# B&R Automation Studio project pneutrunk_plc (part 3)

#### pneutr2_reg_FF_stiff_private.h
```c
/*
 * pneutr2_reg_FF_stiff_private.h
 *
 * Academic License - for use in teaching, academic research, and meeting
 * course requirements at degree granting institutions only.  Not for
 * government, commercial, or other organizational use.
 *
 * Code generation for model "pneutr2_reg_FF_stiff".
 *
 * Model version              : 4.30
 * Simulink Coder version : 9.9 (R2023a) 19-Nov-2022
 * C source code generated on : Thu Feb 15 10:44:02 2024
 *
 * Target selection: bur_grt.tlc
 * Note: GRT includes extra infrastructure and instrumentation for prototyping
 * Embedded hardware selection: Intel->x86/Pentium
 * Code generation objectives: Unspecified
 * Validation result: Not run
 */

#ifndef RTW_HEADER_pneutr2_reg_FF_stiff_private_h_
#define RTW_HEADER_pneutr2_reg_FF_stiff_private_h_
#include "rtwtypes.h"
#include "multiword_types.h"
#include "zero_crossing_types.h"
#include "pneutr2_reg_FF_stiff.h"
#include "pneutr2_reg_FF_stiff_types.h"

extern real32_T look1_tf_binlcpw(real_T u0, const real_T bp0[], const real32_T
  table[], uint32_T maxIndex);
extern void pneutr2_reg_FF_stiff_ID1(real32_T rtu_poz_u_x, real32_T rtu_poz_u_y,
  const real_T rtu_coef_1blue[48], const real_T rtu_coef_2green[48], const
  real_T rtu_coef_3yellow[48], real32_T rtu_tuhost, B_ID1_pneutr2_reg_FF_stiff_T
  *localB);
extern void pneutr2_r_requestedalfa2deltaz1(real32_T rtu_AlphaX_ref, real32_T
  rtu_AlphaY_ref, real32_T rtu_AlphaX_real, real32_T rtu_AlphaY_real, real_T
  rtu_A, real_T rtu_B, real32_T rtu_poradie, B_requestedalfa2deltaz1_pneut_T
  *localB);
extern void pneutr2_reg_FF_s_MATLABFunction(real_T rtu_in, real_T
  rtu_previous_in, real_T rtu_step, real_T rtu_pocet_stepov, real_T rtu_last_in,
  real_T rtu_neupravujuci_uhol, B_MATLABFunction_pneutr2_reg__T *localB);

#endif                          /* RTW_HEADER_pneutr2_reg_FF_stiff_private_h_ */
```

#### pneutr2_reg_FF_stiff_types.h
```c
/*
 * pneutr2_reg_FF_stiff_types.h
 *
 * Academic License - for use in teaching, academic research, and meeting
 * course requirements at degree granting institutions only.  Not for
 * government, commercial, or other organizational use.
 *
 * Code generation for model "pneutr2_reg_FF_stiff".
 *
 * Model version              : 4.30
 * Simulink Coder version : 9.9 (R2023a) 19-Nov-2022
 * C source code generated on : Thu Feb 15 10:44:02 2024
 *
 * Target selection: bur_grt.tlc
 * Note: GRT includes extra infrastructure and instrumentation for prototyping
 * Embedded hardware selection: Intel->x86/Pentium
 * Code generation objectives: Unspecified
 * Validation result: Not run
 */

#ifndef RTW_HEADER_pneutr2_reg_FF_stiff_types_h_
#define RTW_HEADER_pneutr2_reg_FF_stiff_types_h_

/* Forward declaration for rtModel */
typedef struct tag_RTM_pneutr2_reg_FF_stiff_T RT_MODEL_pneutr2_reg_FF_stiff_T;

#endif                            /* RTW_HEADER_pneutr2_reg_FF_stiff_types_h_ */
```

#### rt_nonfinite.h
```c
/*
 * rt_nonfinite.h
 *
 * Academic License - for use in teaching, academic research, and meeting
 * course requirements at degree granting institutions only.  Not for
 * government, commercial, or other organizational use.
 *
 * Code generation for model "pneutr2_reg_FF_stiff".
 *
 * Model version              : 4.30
 * Simulink Coder version : 9.9 (R2023a) 19-Nov-2022
 * C source code generated on : Thu Feb 15 10:44:02 2024
 *
 * Target selection: bur_grt.tlc
 * Note: GRT includes extra infrastructure and instrumentation for prototyping
 * Embedded hardware selection: Intel->x86/Pentium
 * Code generation objectives: Unspecified
 * Validation result: Not run
 */

#ifndef RTW_HEADER_rt_nonfinite_h_
#define RTW_HEADER_rt_nonfinite_h_
#include <stddef.h>
#include "rtwtypes.h"
#define NOT_USING_NONFINITE_LITERALS   1

extern real_T rtInf;
extern real_T rtMinusInf;
extern real_T rtNaN;
extern real32_T rtInfF;
extern real32_T rtMinusInfF;
extern real32_T rtNaNF;
extern void rt_InitInfAndNaN(size_t realSize);
extern boolean_T rtIsInf(real_T value);
extern boolean_T rtIsInfF(real32_T value);
extern boolean_T rtIsNaN(real_T value);
extern boolean_T rtIsNaNF(real32_T value);
typedef struct {
  struct {
    uint32_T wordH;
    uint32_T wordL;
  } words;
} BigEndianIEEEDouble;

typedef struct {
  struct {
    uint32_T wordL;
    uint32_T wordH;
  } words;
} LittleEndianIEEEDouble;

typedef struct {
  union {
    real32_T wordLreal;
    uint32_T wordLuint;
  } wordL;
} IEEESingle;

#endif                                 /* RTW_HEADER_rt_nonfinite_h_ */
```

#### rtGetNaN.h
```c
/*
 * rtGetNaN.h
 *
 * Academic License - for use in teaching, academic research, and meeting
 * course requirements at degree granting institutions only.  Not for
 * government, commercial, or other organizational use.
 *
 * Code generation for model "pneutr2_reg_FF_stiff".
 *
 * Model version              : 4.30
 * Simulink Coder version : 9.9 (R2023a) 19-Nov-2022
 * C source code generated on : Thu Feb 15 10:44:02 2024
 *
 * Target selection: bur_grt.tlc
 * Note: GRT includes extra infrastructure and instrumentation for prototyping
 * Embedded hardware selection: Intel->x86/Pentium
 * Code generation objectives: Unspecified
 * Validation result: Not run
 */

#ifndef RTW_HEADER_rtGetNaN_h_
#define RTW_HEADER_rtGetNaN_h_
#include "rt_nonfinite.h"
#include "rtwtypes.h"

extern real_T rtGetNaN(void);
extern real32_T rtGetNaNF(void);

#endif                                 /* RTW_HEADER_rtGetNaN_h_ */
```

#### rtGetNaN.c
```c
/*
 * rtGetNaN.c
 *
 * Academic License - for use in teaching, academic research, and meeting
 * course requirements at degree granting institutions only.  Not for
 * government, commercial, or other organizational use.
 *
 * Code generation for model "pneutr2_reg_FF_stiff".
 *
 * Model version              : 4.30
 * Simulink Coder version : 9.9 (R2023a) 19-Nov-2022
 * C source code generated on : Thu Feb 15 10:44:02 2024
 *
 * Target selection: bur_grt.tlc
 * Note: GRT includes extra infrastructure and instrumentation for prototyping
 * Embedded hardware selection: Intel->x86/Pentium
 * Code generation objectives: Unspecified
 * Validation result: Not run
 */

#include "rtwtypes.h"
#include "rtGetNaN.h"
#include <stddef.h>
#include "rt_nonfinite.h"
#define NumBitsPerChar                 8U

/*
 * Initialize rtNaN needed by the generated code.
 * NaN is initialized as non-signaling. Assumes IEEE.
 */
real_T rtGetNaN(void)
{
  size_t bitsPerReal = sizeof(real_T) * (NumBitsPerChar);
  real_T nan = 0.0;
  if (bitsPerReal == 32U) {
    nan = rtGetNaNF();
  } else {
    uint16_T one = 1U;
    enum {
      LittleEndian,
      BigEndian
    } machByteOrder = (*((uint8_T *) &one) == 1U) ? LittleEndian : BigEndian;
    switch (machByteOrder) {
     case LittleEndian:
      {
        union {
          LittleEndianIEEEDouble bitVal;
          real_T fltVal;
        } tmpVal;

        tmpVal.bitVal.words.wordH = 0xFFF80000U;
        tmpVal.bitVal.words.wordL = 0x00000000U;
        nan = tmpVal.fltVal;
        break;
      }

     case BigEndian:
      {
        union {
          BigEndianIEEEDouble bitVal;
          real_T fltVal;
        } tmpVal;

        tmpVal.bitVal.words.wordH = 0x7FFFFFFFU;
        tmpVal.bitVal.words.wordL = 0xFFFFFFFFU;
        nan = tmpVal.fltVal;
        break;
      }
    }
  }

  return nan;
}

/*
 * Initialize rtNaNF needed by the generated code.
 * NaN is initialized as non-signaling. Assumes IEEE.
 */
real32_T rtGetNaNF(void)
{
  IEEESingle nanF = { { 0.0F } };

  uint16_T one = 1U;
  enum {
    LittleEndian,
    BigEndian
  } machByteOrder = (*((uint8_T *) &one) == 1U) ? LittleEndian : BigEndian;
  switch (machByteOrder) {
   case LittleEndian:
    {
      nanF.wordL.wordLuint = 0xFFC00000U;
      break;
    }

   case BigEndian:
    {
      nanF.wordL.wordLuint = 0x7FFFFFFFU;
      break;
    }
  }

  return nanF.wordL.wordLreal;
}
```

### Types.typ
```iecst
TYPE
	mech : 	STRUCT
		pozadovany_uhol_y_old : ARRAY[0..6]OF REAL;
		real_uhol_y_kalibrovane : ARRAY[0..6]OF REAL;
		real_uhol_x_kalibrovane : ARRAY[0..6]OF REAL;
		pozadovany_uhol_y : ARRAY[0..6]OF REAL;
		pozadovany_uhol_x : ARRAY[0..6]OF REAL;
		FF_stiffness : ARRAY[0..6]OF REAL;
		PID_P : ARRAY[0..6]OF REAL;
		PID_I : ARRAY[0..6]OF REAL;
		PID_D : ARRAY[0..6]OF REAL;
		PID_N : ARRAY[0..6]OF REAL;
		reset_I_reg : ARRAY[0..6]OF REAL;
		tlak3 : ARRAY[0..6]OF REAL;
		tlak2 : ARRAY[0..6]OF REAL;
		tlak1 : ARRAY[0..6]OF REAL;
		poradie : ARRAY[0..6]OF INT;
		error_total : ARRAY[0..6]OF REAL;
		error_y : ARRAY[0..6]OF REAL;
		error_x : ARRAY[0..6]OF REAL;
		pozadovany_uhol_x_old : ARRAY[0..6]OF REAL;
		nula_y : ARRAY[0..6]OF REAL;
		nula_x : ARRAY[0..6]OF REAL;
		pozadovanyLinear : REAL;
		efektor : BOOL;
	END_STRUCT;
END_TYPE
```

### mem_mgr.h
```c
/*
 * Copyright 1994-2002 The MathWorks, Inc.
 *
 * File: mem_mgr.h
 *
 * Abstract:
 */

#ifndef __MEM_MGR__
#define __MEM_MGR__

struct MemBufHdr {
    struct MemBufHdr *memBufNext;
    struct MemBufHdr *memBufPrev;
    char   *MemBuf;
    int    size;
};

typedef struct MemBufHdr MemBufHdr;

extern void ExtModeFree(void *mem);

extern void *ExtModeMalloc(size_t size);

extern void *ExtModeCalloc(size_t number, size_t size);

#endif /* __MEM_MGR__ */

/* [EOF] mem_mgr.h */
```

### Program Logical/Source/Narazy

#### Cyclic.st
```iecst
PROGRAM _CYCLIC

	FOR i:=0 TO 6 BY 1 DO
		IF modul.naraz[i] = TRUE THEN
			modul.narazAktivny	:= TRUE;
			step				:= 5;
		END_IF
	END_FOR

END_PROGRAM
```

### Program Logical/Source/RS485/Receiver

#### Receiver.typ
```iecst
(********************************************************************
 * COPYRIGHT -- Bernecker + Rainer
 ********************************************************************
 * Program: Receiver
 * File: Receiver.typ
 * Author: Bernecker & Rainer
 * Created: January 25, 2010
 ********************************************************************
 * Local data types of program Receiver
 ********************************************************************)
(*Enumeration for Statemachine*)

TYPE
	enRECV_STEPS :
		(
		FRM_WAIT := 0, (*Defines the wait step*)
		FRM_OPEN, (*Defines Step for FRM_xopen() *)
		FRM_READ, (*Defines Step for FRM_read()*)
		FRM_COPY_RD_DATA, (*Defines Step for storing read data*)
		FRM_RBUF, (*Defines Step for FRM_rbuf()*)
		FRM_CLOSE, (*Defines Step for FRM_close()*)
		FRM_ERROR := 255 (*Defines Step for Errorhandling*)
		);
END_TYPE

(*Command data type*)

TYPE
	command_typ : 	STRUCT
		open_receive : BOOL; (*Open serial port and receive data*)
		close : BOOL; (*Close serial port*)
	END_STRUCT;
END_TYPE

(*Receiver type*)

TYPE
	Receiver_typ : 	STRUCT
		step : enRECV_STEPS; (*Step of the Statemachine*)
		Commands : command_typ; (*Commandinterface*)
		receive_data : ARRAY[0..10]OF BYTE; (*receive data*)
		FRM_xopen_0 : FRM_xopen; (*Functionblock FRM_xopen()*)
		xopenConfig : XOPENCONFIG; (*Configuration Type for FRM_xopen()*)
		FRM_read_0 : FRM_read; (*Functionblock FRM_read()*)
		FRM_rbuf_0 : FRM_rbuf; (*Functionblock FRM_rbuf()*)
		FRM_close_0 : FRM_close; (*Functionblock FRM_close()*)
	END_STRUCT;
END_TYPE
```

#### ReceiverCyclic.st
```iecst
(********************************************************************
 * COPYRIGHT -- Bernecker + Rainer
 ********************************************************************
 * Program: Receiver
 * File: ReceiverCyclic.st
 * Author: Bernecker & Rainer
 * Created: January 25, 2010
 ********************************************************************
 * Implementation of program Receiver
 ********************************************************************)

(*************init program**********************)
PROGRAM _INIT
	Receiver.Commands.open_receive := TRUE;												(*enable Receiver by default*)
END_PROGRAM

(*************cyclic program********************)
PROGRAM _CYCLIC

	CASE Receiver.step OF
		FRM_WAIT:	(*--- wait for command*)

			IF Receiver.Commands.open_receive = TRUE THEN								(*command for Receiver activation*)
				Receiver.step := FRM_OPEN;
   			END_IF

			(*close will be requested in step FRM_RBUF*)

		FRM_OPEN:	(*--- open serial interface*)

			(*Parameters for FRM_xopen()*)
			Receiver.FRM_xopen_0.enable := TRUE;
			Receiver.FRM_xopen_0.device := ADR('IF6.ST1.IF1');							(*Devicename --> see your serial interface properties*)
			Receiver.FRM_xopen_0.mode := ADR('/PHY=RS485 /BD=38400 /DB=8 /PA=N /SB=1'); (*Modestring --> specifies the seria operation mode*)
			Receiver.FRM_xopen_0.config := ADR(Receiver.xopenConfig) ;					(*Additional Parameters, optional*)

			(*Additional Parameters for FRM_xopen()*)
			Receiver.xopenConfig.idle := 10;											(*Idle time between two characters*)
			Receiver.xopenConfig.delimc := 0;											(*activate two delimeters*)
			Receiver.xopenConfig.delim[0] := 0; 										(*e.g. CR - carridge return -> dec 13*)
			Receiver.xopenConfig.delim[1] := 0; 										(*e.g. LF - line feed -> dec 10*)
			Receiver.xopenConfig.tx_cnt := 3;											(*number of transmit buffers*)
			Receiver.xopenConfig.rx_cnt := 3; 											(*number of receive buffers*)
			Receiver.xopenConfig.tx_len := 256; 										(*length of transmit buffers*)
			Receiver.xopenConfig.rx_len := 256; 										(*lenght of receive buffers*)
			Receiver.xopenConfig.argc := 0;												(*activate additional options*)
			Receiver.xopenConfig.argv := 0;												(*parameters for additional options (check help)*)

			Receiver.FRM_xopen_0();														(*call the FRM_xopen() function*)

			IF Receiver.FRM_xopen_0.status = 0 THEN
				Receiver.step := FRM_READ;												(*Interface opend successfully --> next step*)
			ELSIF Receiver.FRM_xopen_0.status = BUSY THEN
				Receiver.step := FRM_OPEN;												(*operation not finished yet --> call again*)
			ELSE
				Receiver.step := FRM_ERROR;												(*function returned errorcode --> check help*)
   			END_IF

		FRM_READ:	(*--- read data from serial interface*)
			Receiver.FRM_read_0.enable := TRUE;
   			Receiver.FRM_read_0.ident := Receiver.FRM_xopen_0.ident;

			Receiver.FRM_read_0();														(*call the FRM_read() function*)

			IF Receiver.FRM_read_0.status = 0 THEN
				Receiver.step := FRM_COPY_RD_DATA;										(*system returned a valid data --> next step*)
			ELSIF Receiver.FRM_read_0.status = frmERR_NOINPUT THEN
				Receiver.step := FRM_READ;												(*no data available --> call again*)
			ELSIF Receiver.FRM_read_0.status = frmERR_INPUTERROR THEN
				Receiver.step := FRM_RBUF;												(*received Frame with defective characters, skip data*)
			ELSE
				Receiver.step := FRM_ERROR;												(*function returned errorcode --> check help*)
   			END_IF

		FRM_COPY_RD_DATA: (*--- copy data out of the receive buffer*)
			(*
			FOR i:=0 TO 8 BY 1 DO
				packet485.packet[i] := Receiver.receive_data[i];
			END_FOR
			*)
			memset(ADR(Receiver.receive_data),0,SIZEOF(Receiver.receive_data));			(*clear read_data buffer*)
			memcpy(ADR(Receiver.receive_data),Receiver.FRM_read_0.buffer,Receiver.FRM_read_0.buflng);     (*copy and evaluate read data*)

			IF(Receiver.receive_data[0] = 255)THEN
				IF(Receiver.receive_data[1] = 255)THEN
					IF(Receiver.receive_data[9] = 254)THEN
						IF(Receiver.receive_data[10] = 254)THEN
							IF(Receiver.receive_data[2] = 1)THEN
								modul.uholINT1 := BYTE_TO_INT(Receiver.receive_data[5]);
								modul.uholINT1 := SHL(modul.uholINT1,8);
								modul.uholINT1  := modul.uholINT1  + BYTE_TO_INT(Receiver.receive_data[6]);
								modul.uhol1[0] := modul.uholINT1;
								modul.uhol1[0] := modul.uhol1[0]*260/1024 - 130;
								modul.uhol1[0] := modul.uhol1[0]*1.0254 + 88.307;
								modul.uholINT2 := BYTE_TO_INT(Receiver.receive_data[7]);
								modul.uholINT2 := SHL(modul.uholINT2,8);
								modul.uholINT2  := modul.uholINT2  + BYTE_TO_INT(Receiver.receive_data[8]);
								modul.uhol2[0] := (modul.uholINT2);
								modul.uhol2[0] := modul.uhol2[0]*260/1024 - 130;
								modul.uhol2[0] := modul.uhol2[0]*1.0254 + 88.307;
							ELSIF(Receiver.receive_data[2] = 2)THEN
								modul.uholINT1 := BYTE_TO_INT(Receiver.receive_data[5]);
								modul.uholINT1 := SHL(modul.uholINT1,8);
								modul.uholINT1  := modul.uholINT1  + BYTE_TO_INT(Receiver.receive_data[6]);
								modul.uhol1[1] := (modul.uholINT1);
								modul.uhol1[1] := modul.uhol1[1]*260/1024 - 130;
								modul.uhol1[1] := modul.uhol1[1]*1.0254 + 88.307;
								modul.uholINT2 := BYTE_TO_INT(Receiver.receive_data[7]);
								modul.uholINT2 := SHL(modul.uholINT2,8);
								modul.uholINT2  := modul.uholINT2  + BYTE_TO_INT(Receiver.receive_data[8]);
								modul.uhol2[1] := (modul.uholINT2);
								modul.uhol2[1] := modul.uhol2[1]*260/1024 - 130;
								modul.uhol2[1] := modul.uhol2[1]*1.0254 + 88.307;
							ELSIF(Receiver.receive_data[2] = 3)THEN
								modul.uholINT1 := BYTE_TO_INT(Receiver.receive_data[5]);
								modul.uholINT1 := SHL(modul.uholINT1,8);
								modul.uholINT1  := modul.uholINT1  + BYTE_TO_INT(Receiver.receive_data[6]);
								modul.uhol1[2] := (modul.uholINT1);
								modul.uhol1[2] := modul.uhol1[2]*260/1024 - 130;
								modul.uhol1[2] := modul.uhol1[2]*1.0254 + 88.307;
								modul.uholINT2 := BYTE_TO_INT(Receiver.receive_data[7]);
								modul.uholINT2 := SHL(modul.uholINT2,8);
								modul.uholINT2  := modul.uholINT2  + BYTE_TO_INT(Receiver.receive_data[8]);
								modul.uhol2[2] := (modul.uholINT2);
								modul.uhol2[2] := modul.uhol2[2]*260/1024 - 130;
								modul.uhol2[2] := modul.uhol2[2]*1.0254 + 88.307;
								IF Receiver.receive_data[4] = 3 THEN
									modul.naraz[2]	:= TRUE;
								ELSE
									modul.naraz[2]	:= FALSE;
								END_IF
							ELSIF(Receiver.receive_data[2] = 4)THEN
								modul.uholINT1 := BYTE_TO_INT(Receiver.receive_data[5]);
								modul.uholINT1 := SHL(modul.uholINT1,8);
								modul.uholINT1  := modul.uholINT1  + BYTE_TO_INT(Receiver.receive_data[6]);
								modul.uhol1[3] := (modul.uholINT1);
								modul.uhol1[3] := modul.uhol1[3]*260/1024 - 130;
								modul.uhol1[3] := modul.uhol1[3]*1.0254 + 88.307;
								modul.uholINT2 := BYTE_TO_INT(Receiver.receive_data[7]);
								modul.uholINT2 := SHL(modul.uholINT2,8);
								modul.uholINT2  := modul.uholINT2  + BYTE_TO_INT(Receiver.receive_data[8]);
								modul.uhol2[3] := (modul.uholINT2);
								modul.uhol2[3] := modul.uhol2[3]*260/1024 - 130;
								modul.uhol2[3] := modul.uhol2[3]*1.0254 + 88.307;
								IF Receiver.receive_data[4] = 3 THEN
									modul.naraz[3]	:= TRUE;
								ELSE
									modul.naraz[3]	:= FALSE;
								END_IF
							ELSIF(Receiver.receive_data[2] = 5)THEN
								modul.uholINT1 := BYTE_TO_INT(Receiver.receive_data[5]);
								modul.uholINT1 := SHL(modul.uholINT1,8);
								modul.uholINT1  := modul.uholINT1  + BYTE_TO_INT(Receiver.receive_data[6]);
								modul.uhol1[4] := (modul.uholINT1);
								modul.uhol1[4] := modul.uhol1[4]*260/1024 - 130;
								modul.uhol1[4] := modul.uhol1[4]*1.0254 + 88.307;
								modul.uholINT2 := BYTE_TO_INT(Receiver.receive_data[7]);
								modul.uholINT2 := SHL(modul.uholINT2,8);
								modul.uholINT2  := modul.uholINT2  + BYTE_TO_INT(Receiver.receive_data[8]);
								modul.uhol2[4] := (modul.uholINT2);
								modul.uhol2[4] := modul.uhol2[4]*260/1024 - 130;
								modul.uhol2[4] := modul.uhol2[4]*1.0254 + 88.307;
								IF Receiver.receive_data[4] = 3 THEN
									modul.naraz[4]	:= TRUE;
								ELSE
									modul.naraz[4]	:= FALSE;
								END_IF
							ELSIF(Receiver.receive_data[2] = 6)THEN
								modul.uholINT1 := BYTE_TO_INT(Receiver.receive_data[5]);
								modul.uholINT1 := SHL(modul.uholINT1,8);
								modul.uholINT1  := modul.uholINT1  + BYTE_TO_INT(Receiver.receive_data[6]);
								modul.uhol1[5] := (modul.uholINT1);
								modul.uhol1[5] := modul.uhol1[5]*260/1024 - 130;
								modul.uhol1[5] := modul.uhol1[5]*1.0254 + 88.307;
								modul.uholINT2 := BYTE_TO_INT(Receiver.receive_data[7]);
								modul.uholINT2 := SHL(modul.uholINT2,8);
								modul.uholINT2  := modul.uholINT2  + BYTE_TO_INT(Receiver.receive_data[8]);
								modul.uhol2[5] := (modul.uholINT2);
								modul.uhol2[5] := modul.uhol2[5]*260/1024 - 130;
								modul.uhol2[5] := modul.uhol2[5]*1.0254 + 88.307;
								IF Receiver.receive_data[4] = 3 THEN
									modul.naraz[5]	:= TRUE;
								ELSE
									modul.naraz[5]	:= FALSE;
								END_IF
							ELSIF(Receiver.receive_data[2] = 7)THEN
								modul.uholINT1 := BYTE_TO_INT(Receiver.receive_data[5]);
								modul.uholINT1 := SHL(modul.uholINT1,8);
								modul.uholINT1  := modul.uholINT1  + BYTE_TO_INT(Receiver.receive_data[6]);
								modul.uhol1[6] := (modul.uholINT1);
								modul.uhol1[6] := modul.uhol1[6]*260/1024 - 130;
								modul.uhol1[6] := modul.uhol1[6]*1.0254 + 88.307;
								modul.uholINT2 := BYTE_TO_INT(Receiver.receive_data[7]);
								modul.uholINT2 := SHL(modul.uholINT2,8);
								modul.uholINT2  := modul.uholINT2  + BYTE_TO_INT(Receiver.receive_data[8]);
								modul.uhol2[6] := (modul.uholINT2);
								modul.uhol2[6] := modul.uhol2[6]*260/1024 - 130;
								modul.uhol2[6] := modul.uhol2[6]*1.0254 + 88.307;
								IF Receiver.receive_data[4] = 1 OR Receiver.receive_data[4] = 2 THEN //lebo dve moduly su zapojene do jednej dosky
									modul.naraz[6]	:= TRUE;
								ELSE
									modul.naraz[6]	:= FALSE;
								END_IF
							ELSIF(Receiver.receive_data[2] = 8)THEN
								IF Receiver.receive_data[4] = 3 THEN
									modul.naraz[7]	:= TRUE;
								ELSE
									modul.naraz[7]	:= FALSE;
								END_IF
							END_IF
						END_IF
					END_IF
				END_IF
			END_IF

			Receiver.step := FRM_RBUF;													(*release read buffer*)

		FRM_RBUF:	(*--- release readbuffer*)

			(*Parameters for FRM_rbuf()*)
			Receiver.FRM_rbuf_0.enable := TRUE;
			Receiver.FRM_rbuf_0.ident := Receiver.FRM_xopen_0.ident;					(*ident from FRM_xopen()*)
			Receiver.FRM_rbuf_0.buffer := Receiver.FRM_read_0.buffer;					(*read buffer*)
			Receiver.FRM_rbuf_0.buflng := Receiver.FRM_read_0.buflng;					(*length of sendbuffer*)

			Receiver.FRM_rbuf_0();														(*call the FRM_rbuf() function*)

			IF Receiver.FRM_rbuf_0.status = 0 THEN
				IF Receiver.Commands.close = TRUE THEN
					Receiver.Commands.open_receive := FALSE;								(*disable command open_send*)
					Receiver.step := FRM_CLOSE;											(*request to close serial port*)
				ELSE
					Receiver.step := FRM_READ;											(*read again*)
				END_IF
			ELSIF Receiver.FRM_rbuf_0.status = BUSY THEN
				Receiver.step := FRM_RBUF;												(*operation not finished yet --> call again*)
			ELSIF Receiver.FRM_rbuf_0.status = frmERR_INVALIDBUFFER THEN
				Receiver.step := FRM_READ;												(*buffer is invalid --> read again*)
			ELSE
				Receiver.step := FRM_ERROR;												(*function returned errorcode --> check help*)
   			END_IF

		FRM_CLOSE:	(*--- close the interface*)
			Receiver.FRM_close_0.enable := TRUE;
   			Receiver.FRM_close_0.ident := Receiver.FRM_xopen_0.ident;					(*ident from FRM_xopen()*)

			Receiver.FRM_close_0();														(*call the FRM_close() function*)

			IF Receiver.FRM_close_0.status = 0 THEN
				Receiver.Commands.close := FALSE;										(*disable close command*)
				Receiver.step := FRM_WAIT;												(*closed interface successfully --> wait step*)
			ELSIF Receiver.FRM_close_0.status = BUSY THEN
				Receiver.step := FRM_CLOSE;												(*operation not finished yet --> call again*)
			ELSE
				Receiver.step := FRM_ERROR;												(*function returned errorcode --> check help*)
			END_IF

		FRM_ERROR:	(*--- error handling*)
			; (*not implementet yet, check help for error codes*)
 	END_CASE

END_PROGRAM
```

### Program Logical/Source/RS485/Sender

#### SenderCyclic.st
```iecst
(********************************************************************
 * COPYRIGHT -- Bernecker + Rainer
 ********************************************************************
 * Program: Sender
 * File: SenderCyclic.st
 * Author: Bernecker & Rainer
 * Created: January 25, 2010
 ********************************************************************
 * Implementation of program Sender
 ********************************************************************)

(*************init program**********************)
PROGRAM _INIT
	Sender.Commands.open_send := TRUE;												(*enable sender by default*)
	packet485.sendPacketFinal[0] := 255;
	packet485.sendPacketFinal[1] := 255;
	packet485.sendPacketFinal[2] := 1;				// ID
	packet485.sendPacketFinal[3] := 1;
	packet485.sendPacketFinal[4] := 254;
	packet485.sendPacketFinal[5] := 254;
	Sender.step					 := FRM_WAIT;
END_PROGRAM

(*************cyclic program********************)
PROGRAM _CYCLIC

	CASE Sender.step OF
		FRM_WAIT:	(*--- wait for command*)

			IF Sender.Commands.open_send = TRUE THEN								(*command for sender activation*)
				Sender.step := FRM_OPEN;
   			END_IF

			(*close will be requested in step FRM_WRITE*)

		FRM_OPEN:	(*--- open serial interface*)

			(*Parameters for FRM_xopen()*)
			Sender.FRM_xopen_0.enable := TRUE;
			Sender.FRM_xopen_0.device := ADR('IF6.ST1.IF1');										(*Devicename --> see your serial interface properties*)
			Sender.FRM_xopen_0.mode := ADR('/PHY=RS485 /BD=38400 /DB=8 /PA=N /SB=1'); 		(*Modestring --> specifies the seria operation mode*)
			Sender.FRM_xopen_0.config := ADR(Sender.xopenConfig) ;					(*Additional Parameters, optional*)

			(*Additional Parameters for FRM_xopen()*)
			Sender.xopenConfig.idle := 10;											(*Idle time between two characters*)
			Sender.xopenConfig.delimc := 0;											(*activate two delimeters*)
			Sender.xopenConfig.delim[0] := 0; 										(*CR - carridge return -> dec 13*)
			Sender.xopenConfig.delim[1] := 0; 										(*LF - line feed -> dec 10*)
			Sender.xopenConfig.tx_cnt := 3;											(*number of transmit buffers*)
			Sender.xopenConfig.rx_cnt := 3; 										(*number of receive buffers*)
			Sender.xopenConfig.tx_len := 256; 										(*length of transmit buffers*)
			Sender.xopenConfig.rx_len := 256; 										(*lenght of receive buffers*)
			Sender.xopenConfig.argc := 0;											(*activate additional options*)
			Sender.xopenConfig.argv := 0;											(*parameters for additional options (check help)*)

			Sender.FRM_xopen_0();													(*call the FRM_xopen() function*)

			IF Sender.FRM_xopen_0.status = 0 THEN
				Sender.step := FRM_GBUF;											(*Interface opend successfully --> next step*)
			ELSIF Sender.FRM_xopen_0.status = BUSY THEN
				Sender.step := FRM_OPEN;											(*operation not finished yet --> call again*)
			ELSE
				Sender.step := FRM_ERROR;											(*function returned errorcode --> check help*)
   			END_IF

		FRM_GBUF:	(*--- aquire sendbuffer for FRM_WRITE*)
			Sender.FRM_gbuf_0.enable := TRUE;
   			Sender.FRM_gbuf_0.ident := Sender.FRM_xopen_0.ident;

			Sender.FRM_gbuf_0();													(*call the FRM_gbuf() function*)

			IF Sender.FRM_gbuf_0.status = 0 THEN
				memset(Sender.FRM_gbuf_0.buffer,0,Sender.FRM_gbuf_0.buflng);		(*clear sendbuffer*)
				Sender.step := FRM_PREPARE_SENDDATA;								(*system returned a valid buffer --> next step*)
			ELSIF Sender.FRM_gbuf_0.status = BUSY THEN
				Sender.step := FRM_GBUF;											(*operation not finished yet --> call again*)
			ELSE
				Sender.step := FRM_ERROR;											(*function returned errorcode --> check help*)
   			END_IF

		FRM_PREPARE_SENDDATA: (*--- prepare senddata, copy data to sendbuffer*)

			IF packet485.id = 7 THEN
				packet485.id := 1;
			ELSE
				packet485.id := packet485.id + 1;
			END_IF
			Sender.Commands.open_send := TRUE;										(*enable sender by default*)
			packet485.sendPacketFinal[0] := 255;
			packet485.sendPacketFinal[1] := 255;
			packet485.sendPacketFinal[2] := USINT_TO_BYTE(packet485.id);
			packet485.sendPacketFinal[3] := 1;
			packet485.sendPacketFinal[4] := 254;
			packet485.sendPacketFinal[5] := 254;
			packet485.sendPacketFinal[0] := 255;

			strcpy(Sender.FRM_gbuf_0.buffer,ADR(packet485.sendPacketFinal));		(*copy senddata to sendbuffer*)
			Sender.step := FRM_WRITE;												(*--> next step*)

		FRM_WRITE:	(*--- write data to interface*)

			(*Parameters for FRM_write()*)
			Sender.FRM_write_0.enable := TRUE;
			Sender.FRM_write_0.ident := Sender.FRM_xopen_0.ident;					(*ident from FRM_xopen()*)
			Sender.FRM_write_0.buffer := Sender.FRM_gbuf_0.buffer;					(*sendbuffer*)
			Sender.FRM_write_0.buflng := strlen(ADR(packet485.sendPacketFinal));				(*net length of senddata*)

			Sender.FRM_write_0();													(*call the FRM_write() function*)

			IF Sender.FRM_write_0.status = 0 THEN
				IF Sender.Commands.close = TRUE THEN								(*requst to close the serial port*)
					Sender.Commands.open_send := FALSE;								(*disable command open_send*)
					Sender.step := FRM_CLOSE;
				ELSE
					Sender.step := FRM_GBUF;										(*writing successful --> get next sendbuffer*)
				END_IF
			ELSIF Sender.FRM_write_0.status = BUSY THEN
				Sender.step := FRM_WRITE;											(*operation not finished yet --> call again*)
			ELSE
				Sender.step := FRM_ROBUF;											(*function returned errorcode --> check help*)
   			END_IF

		FRM_ROBUF:	(*--- release sendbuffer in case of no successful write operation*)
			Sender.FRM_robuf_0.enable := TRUE;
			Sender.FRM_robuf_0.buffer := Sender.FRM_gbuf_0.buffer;					(*sendbuffer*)
			Sender.FRM_robuf_0.buflng := Sender.FRM_gbuf_0.buflng;					(*buffer length*)
			Sender.FRM_robuf_0.ident := Sender.FRM_xopen_0.ident;					(*ident open*)

			Sender.FRM_robuf_0();													(*call the FRM_robuf() function*)

			IF Sender.FRM_robuf_0.status = 0 THEN
				Sender.step := FRM_GBUF;											(*released buffer successful --> get next sendbuffer*)
			ELSIF Sender.FRM_robuf_0.status = BUSY THEN
				Sender.step := FRM_ROBUF;											(*operation not finished yet --> call again*)
			ELSE
				Sender.step := FRM_ERROR;											(*function returned errorcode --> check help*)
   			END_IF

		FRM_CLOSE:	(*--- close the interface*)
			Sender.FRM_close_0.enable := TRUE;
   			Sender.FRM_close_0.ident := Sender.FRM_xopen_0.ident;					(*ident from FRM_xopen()*)

			Sender.FRM_close_0();													(*call the FRM_close() function*)

			IF Sender.FRM_close_0.status = 0 THEN
				Sender.Commands.close := FALSE;										(*disable close command*)
				Sender.step := FRM_WAIT;											(*closed interface successfully --> wait step*)
			ELSIF Sender.FRM_close_0.status = BUSY THEN
				Sender.step := FRM_CLOSE;											(*operation not finished yet --> call again*)
			ELSE
				Sender.step := FRM_ERROR;											(*function returned errorcode --> check help*)
			END_IF

		FRM_ERROR:	(*--- error handling*)
			Sender.step := FRM_WAIT;
			//; (*not implementet yet, check help for error codes*)
 	END_CASE

END_PROGRAM
```

### Program Logical/Source/UDP/Client (IEC) - AsUDP Client Application

#### Client.typ
```iecst
(********************************************************************
 * COPYRIGHT -- Bernecker + Rainer
 ********************************************************************
 * Program: Client
 * File: Client.typ
 * Author: Bernecker + Rainer
 * Created: June 02, 2008
 ********************************************************************
 * Local data types of program Client
 ********************************************************************)

TYPE
	Client_typ : 	STRUCT  (*UDP Client Variables*)
		sStep : UINT; (*UDP Client Step Variable*)
		server_address : STRING[20]; (*Address of the Server*)
		server_portnumber : UINT; (*Portnumber of the Server*)
		no_data_received_count : UINT; (*Counts up if no data are received*)
		UdpOpen_0 : UdpOpen; (*AsUDP.UdpOpen FUB*)
		UdpConnect_0 : UdpConnect; (*AsUDP.UdpConnect FUB*)
		UdpSend_0 : UdpSend; (*AsUDP.UdpSend FUB*)
		UdpRecv_0 : UdpRecv; (*AsUDP.UdpRecv FUB*)
		UdpDisconnect_0 : UdpDisconnect; (*AsUDP.UdpDisconnect FUB*)
		UdpClose_0 : UdpClose; (*AsUDP.UdpClose FUB*)
		sendBuffer : STRING[255];
		tempString : STRING[50];
	END_STRUCT;
END_TYPE
```

#### Client.var
```iecst
(********************************************************************
 * COPYRIGHT -- Bernecker + Rainer
 ********************************************************************
 * Program: Client
 * File: Client.var
 * Author: Bernecker + Rainer
 * Created: June 02, 2008
 ********************************************************************
 * Local variables of program Client
 ********************************************************************)
VAR
	Client : Client_typ := (0); (*Data for Client Task*)
	i : INT;
	helpString : STRING[40];
	sendBuffer : BOOL;
	a : INT;
END_VAR
```

#### Client.st
```iecst
(********************************************************************
 * COPYRIGHT -- Bernecker + Rainer
 ********************************************************************
 * Program: Client
 * File: Client.st
 * Author: Bernecker + Rainer
 * Created: June 02, 2008
 ********************************************************************
 * Implementation of program Client
 ********************************************************************)

PROGRAM _CYCLIC

	memset(ADR(Client.sendBuffer),0,SIZEOF(Client.tempString));

	strcat(ADR(Client.sendBuffer),ADR('UhlyX:'));
	FOR i:=0 TO 6 BY 1 DO
		ftoa(modul.uhol1[i],ADR(Client.tempString));
		strcat(ADR(Client.sendBuffer),ADR(Client.tempString));
		IF i < 6 THEN
			strcat(ADR(Client.sendBuffer),ADR(','));
		END_IF
	END_FOR

	strcat(ADR(Client.sendBuffer),ADR(',UhlyY:'));
	FOR i:=0 TO 6 BY 1 DO
		ftoa(modul.uhol2[i],ADR(Client.tempString));
		strcat(ADR(Client.sendBuffer),ADR(Client.tempString));
		IF i < 6 THEN
			strcat(ADR(Client.sendBuffer),ADR(','));
		END_IF
	END_FOR

	strcat(ADR(Client.sendBuffer),ADR(',Narazy:'));
	FOR i:=0 TO 6 BY 1 DO
		itoa(modul.naraz[i],ADR(Client.tempString));
		strcat(ADR(Client.sendBuffer),ADR(Client.tempString));
		IF i < 6 THEN
			strcat(ADR(Client.sendBuffer),ADR(','));
		END_IF
	END_FOR

	//FOR i:=0 TO 6 BY 1 DO
		//ftoa(modul.uhol_XminusRef[i], ADR(helpString));
		//strcat(ADR(LibAsUDP1_ST.send_data), ADR(helpString));
		//strcat(ADR(LibAsUDP1_ST.send_data), ADR(','));
		//(modul.uhol_YminusRef[i], ADR(helpString));
		//strcat(ADR(LibAsUDP1_ST.send_data), ADR(helpString));
		//strcat(ADR(LibAsUDP1_ST.send_data), ADR(','));
	//END_FOR

	//LibAsUDP1_ST.send_data[0] := LibAsUDP1_ST.send_data[0] + 1;  (* Generate a "running" variable for Data transfer *)
	//LibAsUDP1_ST.send_data := '20.12 12.54 10.24 -13.25';

	//memset(ADR(LibAsUDP1_ST.send_data), 0, SIZEOF(LibAsUDP1_ST.send_data));
	//memset(ADR(helpString), 0, SIZEOF(helpString));

	//ftoa(modul.linearReal, ADR(helpString)); // vymenit za linearny
	//strcat(ADR(LibAsUDP1_ST.send_data), ADR(helpString));
	//strcat(ADR(LibAsUDP1_ST.send_data), ADR(','));

	(*
	memset(ADR(LibAsUDP1_ST.send_data), 0, SIZEOF(LibAsUDP1_ST.send_data));
	memset(ADR(helpString), 0, SIZEOF(helpString));

	FOR i:=0 TO 5 BY 1 DO
		ftoa(modul.uhol1[i], ADR(helpString));
		strcat(ADR(LibAsUDP1_ST.send_data), ADR(helpString));
		strcat(ADR(LibAsUDP1_ST.send_data), ADR(','));
		ftoa(modul.uhol2[i], ADR(helpString));
		strcat(ADR(LibAsUDP1_ST.send_data), ADR(helpString));
		strcat(ADR(LibAsUDP1_ST.send_data), ADR(','));
	END_FOR
	ftoa(modul.uhol2[0], ADR(helpString)); // vymenit za linearny
	strcat(ADR(LibAsUDP1_ST.send_data), ADR(helpString));
	//strcat(ADR(LibAsUDP1_ST.send_data), ADR(','));
	*)
	CASE Client.sStep OF

		0:	(* Open UDP Port *)
			Client.UdpOpen_0.enable := 1;
			Client.UdpOpen_0.pIfAddr := 0;	(* Listen on all TCP/IP Interfaces*)
			Client.UdpOpen_0.port := 12051;	(* Port to listen*)
			Client.UdpOpen_0.options := 0;
			Client.UdpOpen_0;	(* Call the Function*)

			IF Client.UdpOpen_0.status = 0 THEN  (* UdpOpen successful*)
				Client.sStep := 1;
			ELSIF Client.UdpOpen_0.status = ERR_FUB_BUSY THEN  (* UdpOpen not finished -> redo *)
			  (* Busy *)
			ELSE  (* Goto Error Step *)
				Client.sStep := 10;
			END_IF

		1:	(* Send Data to the Server *)
			Client.server_address := '192.168.1.88';	(* IP Address of the Server *)
			Client.server_portnumber := 12050;	(* Port number of the Server *)

			Client.UdpSend_0.enable := 1;
			Client.UdpSend_0.ident := Client.UdpOpen_0.ident;	(* Connection Ident from AsUDP.UDP_Open *)
			Client.UdpSend_0.pHost := ADR(Client.server_address);
			Client.UdpSend_0.port := Client.server_portnumber;
			Client.UdpSend_0.pData := ADR(Client.sendBuffer);	(* Which data to send *)
			Client.UdpSend_0.datalen := SIZEOF(Client.sendBuffer);	(* Lenght of data to send *)
			Client.UdpSend_0.flags := 0;
			Client.UdpSend_0;	(* Call the Function*)

			IF Client.UdpSend_0.status = 0 THEN  (* Data sent *)
				Client.sStep := 2;
			ELSIF Client.UdpSend_0.status = ERR_FUB_BUSY THEN  (* UdpSend not finished -> redo *)
			  (* Busy *)
			ELSE  (* Goto Error Step *)
				Client.sStep := 10;
			END_IF

		2:	(* Receive Data from the Server *)
			Client.UdpRecv_0.enable := 1;
			Client.UdpRecv_0.ident := Client.UdpOpen_0.ident;  (* Connection Ident from AsUDP.UDP_Open *)
			Client.UdpRecv_0.pData	:= ADR(LibAsUDP1_ST.receive_data);  (* Where to store the incoming data *)//ADR(LibAsUDP1_ST.receive_data);
			Client.UdpRecv_0.datamax := SIZEOF(LibAsUDP1_ST.receive_data);  (* Lenght of data buffer *)
			Client.UdpRecv_0.flags := 0;
			Client.UdpRecv_0;  (* Call the Function*)

			IF Client.UdpRecv_0.status = 0 THEN  (* Data was received successfully -> Send next packet *)
				Client.sStep := 3;
				Client.no_data_received_count := 0;
			ELSIF Client.UdpRecv_0.status = udpERR_NO_DATA THEN  (* No data received - wait *)
			  (* No Data received *)
			  	Client.no_data_received_count := Client.no_data_received_count + 1;	(* Increase if no data are received *)

				IF Client.no_data_received_count > 200 THEN		(* No data timeout for TC1 [10ms] *)
					Client.no_data_received_count := 0;
					Client.sStep := 1;	(* Send again *)
				END_IF
			ELSIF Client.UdpRecv_0.status = ERR_FUB_BUSY THEN  (* UdpRecv not finished -> redo *)
			  (* Busy *)
			ELSE  (* Goto Error Step *)
				Client.sStep := 10;
			END_IF

		3: (* Close connection *)
			Client.UdpClose_0.enable := 1;
			Client.UdpClose_0.ident := Client.UdpOpen_0.ident;  (* Connection Ident from AsUDP.UDP_Open *)
			Client.UdpClose_0;  (* Call the Function*)

			IF Client.UdpClose_0.status = 0 THEN  (* Close successful -> Reopen the interface *)
				Client.sStep := 0;
			ELSIF Client.UdpClose_0.status = ERR_FUB_BUSY THEN  (* UdpClose not finished -> redo *)
			  (* Busy *)
			ELSE  (* Goto Error Step *)
				Client.sStep := 10;
			END_IF

		10: (* Here some error Handling has to be implemented *)

	END_CASE

END_PROGRAM
```

### Program Logical/Source/UDP/Server (IEC) - AsUDP Server Application

#### Server.typ
```iecst
(********************************************************************
 * COPYRIGHT -- Bernecker + Rainer
 ********************************************************************
 * Program: Server
 * File: Server.typ
 * Author: Bernecker + Rainer
 * Created: June 02, 2008
 ********************************************************************
 * Local data types of program Server
 ********************************************************************)

TYPE
	Server_typ : 	STRUCT  (*UDP Server Variables*)
		sStep : UINT; (*UDP Server Step Variable*)
		client_address : STRING[20]; (*Address of the client connection to the Server*)
		UdpOpen_0 : UdpOpen; (*AsUDP.UdpOpen FUB*)
		UdpConnect_0 : UdpConnect; (*AsUDP.UdpConnect FUB*)
		UdpSend_0 : UdpSend; (*AsUDP.UdpSend FUB*)
		UdpRecv_0 : UdpRecv; (*AsUDP.UdpRecv FUB*)
		UdpDisconnect_0 : UdpDisconnect; (*AsUDP.UdpDisconnect FUB*)
		UdpClose_0 : UdpClose; (*AsUDP.UdpClose FUB*)
		data_buffer : STRING[256]; (*Data buffer ( receive and send )*)
	END_STRUCT;
END_TYPE
```

#### Server.var
```iecst
(********************************************************************
 * COPYRIGHT -- Bernecker + Rainer
 ********************************************************************
 * Program: Server
 * File: Server.var
 * Author: Bernecker + Rainer
 * Created: June 02, 2008
 ********************************************************************
 * Local variables of program Server
 ********************************************************************)
VAR
	Server : Server_typ := (0); (*Data for Server Task*)
	i : INT;
	switch : BOOL;
	Pa : INT;
	a : INT;
END_VAR
```

#### Server.st
```iecst
(********************************************************************
 * COPYRIGHT -- Bernecker + Rainer
 ********************************************************************
 * Program: Server
 * File: Server.st
 * Author: Bernecker + Rainer
 * Created: June 02, 2008
 ********************************************************************
 * Implementation of program Server
 ********************************************************************)

PROGRAM _CYCLIC

	CASE Server.sStep OF

		0:	(* Open UDP Port *)
			Server.UdpOpen_0.enable := 1;
			Server.UdpOpen_0.pIfAddr := 0;	(* Listen on all TCP/IP Interfaces*)
			Server.UdpOpen_0.port := 12050;	(* Port to listen*)
			Server.UdpOpen_0.options := 0;
			Server.UdpOpen_0;	(* Call the Function*)

			IF Server.UdpOpen_0.status = 0 THEN  (* UdpOpen successful*)
				Server.sStep := 1;
			ELSIF Server.UdpOpen_0.status = ERR_FUB_BUSY THEN  (* UdpOpen not finished -> redo *)
			  (* Busy *)
			ELSE  (* Goto Error Step *)
				Server.sStep := 10;
			END_IF

		1:	(* Wait for Data *)
			Server.UdpRecv_0.enable := 1;
			Server.UdpRecv_0.ident := Server.UdpOpen_0.ident;	(* Client Ident from AsUDP.UDP_Open *)
			Server.UdpRecv_0.pData := ADR(Server.data_buffer);	(* Where to store the incoming data *)
			Server.UdpRecv_0.datamax := SIZEOF(Server.data_buffer);	(* Lenght of data buffer *)
			Server.UdpRecv_0.flags := 0;
			Server.UdpRecv_0.pIpAddr := ADR(Server.client_address);	(* IP Address of the Client *)
			Server.UdpRecv_0;	(* Call the Function*)

			IF Server.UdpRecv_0.status = 0 THEN  (* Data received *)
				Server.sStep := 2;
			ELSIF Server.UdpRecv_0.status = udpERR_NO_DATA THEN  (* No data received - wait *)
			  (* No Data received *)
			ELSIF Server.UdpRecv_0.status = ERR_FUB_BUSY THEN  (* UdpRecv not finished -> redo *)
			  (* Busy *)
			ELSE  (* Goto Error Step *)
				Server.sStep := 10;
			END_IF

		2:	(* Send Data back to Client *)

			Server.UdpSend_0.enable := 1;
			Server.UdpSend_0.ident := Server.UdpOpen_0.ident;	// Client Ident from AsUDP.UDP_Open
			Server.UdpSend_0.pHost := ADR(Server.client_address);	// IP Address of the Client
			Server.UdpSend_0.port := Server.UdpRecv_0.port;		// Port number of the Client
			Server.UdpSend_0.pData := ADR(Server.data_buffer);	// Which data to send
			Server.UdpSend_0.datalen := SIZEOF(Server.data_buffer);	// Lenght of data to send
			Server.UdpSend_0.flags := 0;
			Server.UdpSend_0;	// Call the Function

			IF switch = FALSE THEN
				// Yellow - 1, Red - 2, Undefined - 3
				packetPos.color := FIND(Server.data_buffer, 'yellow');
				IF(packetPos.color>1)THEN
					automatika.step_color := 1;
				ELSIF(packetPos.color=0)THEN
					packetPos.color := FIND(Server.data_buffer, 'red');
					IF(packetPos.color>1) THEN
						automatika.step_color:= 2;
					ELSE
						automatika.step_color:= 3;
					END_IF

				END_IF
				// Volba kroku robota
				packetPos.step := FIND(Server.data_buffer, 'come');
				IF(packetPos.step >1)THEN
					global_step_udp := 1;
				ELSIF(packetPos.step = 0)THEN
					packetPos.step := FIND(Server.data_buffer, 'hold');
					IF(packetPos.step >1)THEN
						global_step_udp := 2;
					ELSIF(packetPos.step = 0)THEN
						packetPos.step := FIND(Server.data_buffer, 'release');
						IF(packetPos.step >1)THEN
							global_step_udp := 3;
						ELSIF(packetPos.step = 0)THEN
							packetPos.step := FIND(Server.data_buffer, 'continue');
							IF(packetPos.step >1)THEN
								global_step_udp := 4;
							END_IF
						END_IF
					END_IF
				END_IF

				packetPos.tlak1pos := FIND(Server.data_buffer, 'tlak1:');
				packetPos.tlak2pos := FIND(Server.data_buffer, 'tlak2:');
				packetPos.tlak3pos := FIND(Server.data_buffer, 'tlak3:');
				packetPos.end := FIND(Server.data_buffer, 'end');

				packetPos.tlak1Full := MID(Server.data_buffer, packetPos.tlak2pos - packetPos.tlak1pos -6,packetPos.tlak1pos+6);
				packetPos.tlak2Full := MID(Server.data_buffer, packetPos.tlak3pos - packetPos.tlak2pos -6,packetPos.tlak2pos +6);
				packetPos.tlak3Full := MID(Server.data_buffer, packetPos.end - packetPos.tlak3pos -6,packetPos.tlak3pos +6);

				FOR i:=0 TO 6 BY 1 DO	//11
					packetPos.commatlak1 := FIND(packetPos.tlak1Full, ',');
					packetPos.tlak1String[i] := MID(packetPos.tlak1Full, packetPos.commatlak1, 0);
					packetPos.tlak1Full := DELETE(packetPos.tlak1Full,packetPos.commatlak1+1, 0);
					packetPos.tlak1Desired[i] := atof(ADR(packetPos.tlak1String[i])) ;
					IF packetPos.tlak1Desired[i] >= packetPos.MAX_VALUE THEN
						packetPos.tlak1Desired[i] := packetPos.MAX_VALUE;
					END_IF
					modul.tlak1[i] := REAL_TO_INT(packetPos.tlak1Desired[i]);
				END_FOR

				FOR i:=0 TO 6 BY 1 DO	//11
					packetPos.commatlak2 := FIND(packetPos.tlak2Full, ',');
					packetPos.tlak2String[i] := MID(packetPos.tlak2Full, packetPos.commatlak2, 0);
					packetPos.tlak2Full := DELETE(packetPos.tlak2Full,packetPos.commatlak2+1, 0);
					packetPos.tlak2Desired[i] := atof(ADR(packetPos.tlak2String[i])) ;
					IF packetPos.tlak2Desired[i] >= packetPos.MAX_VALUE THEN
						packetPos.tlak2Desired[i] := packetPos.MAX_VALUE;
					END_IF
					modul.tlak2[i] := REAL_TO_INT(packetPos.tlak2Desired[i]);
				END_FOR

				FOR i:=0 TO 6 BY 1 DO	//11
					packetPos.commatlak3 := FIND(packetPos.tlak3Full, ',');
					packetPos.tlak3String[i] := MID(packetPos.tlak3Full, packetPos.commatlak3, 0);
					packetPos.tlak3Full := DELETE(packetPos.tlak3Full,packetPos.commatlak3+1, 0);
					packetPos.tlak3Desired[i] := atof(ADR(packetPos.tlak3String[i])) ;
					IF packetPos.tlak3Desired[i] >= packetPos.MAX_VALUE THEN
						packetPos.tlak3Desired[i] := packetPos.MAX_VALUE;
					END_IF
					modul.tlak3[i] := REAL_TO_INT(packetPos.tlak3Desired[i]);
				END_FOR

				(*FOR i:= 0 TO 6 BY 1 DO
					IF packetPos.tlak2Desired[i] >= packetPos.MAX_VALUE THEN
						packetPos.tlak2Desired[i] := packetPos.MAX_VALUE;
						modul.tlak2[i] := REAL_TO_INT(packetPos.tlak2Desired[i]);
					END_IF;
			    END_FOR *)

				//modul.tlak2[i] := REAL_TO_INT(packetPos.tlak2Desired[i]);
				// Server.data_buffer bolo povodne ked to slo STRING[5][0..100] a tu bolo Server.data_buffer[0]
				(*packetPos.p := FIND(Server.data_buffer, 'p:');
				packetPos.alpha := FIND(Server.data_buffer, 'a:');
				packetPos.end := FIND(Server.data_buffer, 'end');
				packetPos.pLength := UDINT_TO_INT(Server.UdpSend_0.datalen) - (packetPos.p + 1) - packetPos.alpha;
				packetPos.pFull := MID(Server.data_buffer, packetPos.alpha - packetPos.p -2,packetPos.p +2);
				packetPos.alphaLength := UDINT_TO_INT(Server.UdpSend_0.datalen) - (packetPos.alpha - 1) - packetPos.p;
				packetPos.alphaFull := MID(Server.data_buffer, packetPos.end+2 - packetPos.alpha, packetPos.alpha+2);

				packetPos.alphaFull := MID(Server.data_buffer, 13, 19);
				packetPos.alphaFullinfo:=packetPos.alphaFull;
				packetPos.pFullinfo:=packetPos.pFull;
				FOR i:=0 TO 3 BY 1 DO	//11
					packetPos.commaP := FIND(packetPos.pFull, ',');
					packetPos.pString[i] := MID(packetPos.pFull, packetPos.commaP, 0);
					packetPos.pFull := DELETE(packetPos.pFull,packetPos.commaP+1, 0);
					packetPos.pDesired[i] := atof(ADR(packetPos.pString[i])) ;
				END_FOR

				FOR a:=0 TO 3 BY 1 DO
				packetPos.commaAlpha := FIND(packetPos.alphaFull, ',');
				packetPos.alphaString[a] := MID(packetPos.alphaFull, packetPos.commaAlpha, 0);
				//modul.tlaky[a]:=atof(ADR(packetPos.alphaString[a])) ;
				packetPos.alphaFull := DELETE(packetPos.alphaFull,packetPos.commaAlpha+1, 0);
				packetPos.alphaDesired[a] := atof(ADR(packetPos.alphaString[a])) ;
				END_FOR*)

				//packetPos.pString[3] := MID(packetPos.qFull, packetPos.comma, 0);//12
				//packetPos.qFull := DELETE(packetPos.qFull, packetPos.comma+1, 0);
				//packetPos.qDesired[14] := atof(ADR(packetPos.qString[14]));//12
			END_IF

			IF Server.UdpSend_0.status = 0 THEN  (* Data sent *)
				Server.sStep := 1;
			ELSIF Server.UdpSend_0.status = ERR_FUB_BUSY THEN  (* UdpSend not finished -> redo *)
				(* Busy *)
			ELSE  (* Goto Error Step *)
				Server.sStep := 10;
			END_IF

		10:  (* Here some error Handling has to be implemented *)

	END_CASE

END_PROGRAM
```

### Program Logical/test_input

#### rt_nonfinite.h
```c
/*
 * rt_nonfinite.h
 *
 * Academic License - for use in teaching, academic research, and meeting
 * course requirements at degree granting institutions only.  Not for
 * government, commercial, or other organizational use.
 *
 * Code generation for model "simulink_2_plc".
 *
 * Model version              : 1.4
 * Simulink Coder version : 9.9 (R2023a) 19-Nov-2022
 * C source code generated on : Tue Feb  6 09:08:04 2024
 *
 * Target selection: bur_grt.tlc
 * Note: GRT includes extra infrastructure and instrumentation for prototyping
 * Embedded hardware selection: Intel->x86/Pentium
 * Code generation objectives: Unspecified
 * Validation result: Not run
 */

#ifndef RTW_HEADER_rt_nonfinite_h_
#define RTW_HEADER_rt_nonfinite_h_
#include <stddef.h>
#include "rtwtypes.h"
#define NOT_USING_NONFINITE_LITERALS   1

extern real_T rtInf;
extern real_T rtMinusInf;
extern real_T rtNaN;
extern real32_T rtInfF;
extern real32_T rtMinusInfF;
extern real32_T rtNaNF;
extern void rt_InitInfAndNaN(size_t realSize);
extern boolean_T rtIsInf(real_T value);
extern boolean_T rtIsInfF(real32_T value);
extern boolean_T rtIsNaN(real_T value);
extern boolean_T rtIsNaNF(real32_T value);
typedef struct {
  struct {
    uint32_T wordH;
    uint32_T wordL;
  } words;
} BigEndianIEEEDouble;

typedef struct {
  struct {
    uint32_T wordL;
    uint32_T wordH;
  } words;
} LittleEndianIEEEDouble;

typedef struct {
  union {
    real32_T wordLreal;
    uint32_T wordLuint;
  } wordL;
} IEEESingle;

#endif                                 /* RTW_HEADER_rt_nonfinite_h_ */
```

#### rtGetNaN.c
```c
/*
 * rtGetNaN.c
 *
 * Academic License - for use in teaching, academic research, and meeting
 * course requirements at degree granting institutions only.  Not for
 * government, commercial, or other organizational use.
 *
 * Code generation for model "simulink_2_plc".
 *
 * Model version              : 1.4
 * Simulink Coder version : 9.9 (R2023a) 19-Nov-2022
 * C source code generated on : Tue Feb  6 09:08:04 2024
 *
 * Target selection: bur_grt.tlc
 * Note: GRT includes extra infrastructure and instrumentation for prototyping
 * Embedded hardware selection: Intel->x86/Pentium
 * Code generation objectives: Unspecified
 * Validation result: Not run
 */

#include "rtwtypes.h"
#include "rtGetNaN.h"
#include <stddef.h>
#include "rt_nonfinite.h"
#define NumBitsPerChar                 8U

/*
 * Initialize rtNaN needed by the generated code.
 * NaN is initialized as non-signaling. Assumes IEEE.
 */
real_T rtGetNaN(void)
{
  size_t bitsPerReal = sizeof(real_T) * (NumBitsPerChar);
  real_T nan = 0.0;
  if (bitsPerReal == 32U) {
    nan = rtGetNaNF();
  } else {
    uint16_T one = 1U;
    enum {
      LittleEndian,
      BigEndian
    } machByteOrder = (*((uint8_T *) &one) == 1U) ? LittleEndian : BigEndian;
    switch (machByteOrder) {
     case LittleEndian:
      {
        union {
          LittleEndianIEEEDouble bitVal;
          real_T fltVal;
        } tmpVal;

        tmpVal.bitVal.words.wordH = 0xFFF80000U;
        tmpVal.bitVal.words.wordL = 0x00000000U;
        nan = tmpVal.fltVal;
        break;
      }

     case BigEndian:
      {
        union {
          BigEndianIEEEDouble bitVal;
          real_T fltVal;
        } tmpVal;

        tmpVal.bitVal.words.wordH = 0x7FFFFFFFU;
        tmpVal.bitVal.words.wordL = 0xFFFFFFFFU;
        nan = tmpVal.fltVal;
        break;
      }
    }
  }

  return nan;
}

/*
 * Initialize rtNaNF needed by the generated code.
 * NaN is initialized as non-signaling. Assumes IEEE.
 */
real32_T rtGetNaNF(void)
{
  IEEESingle nanF = { { 0.0F } };

  uint16_T one = 1U;
  enum {
    LittleEndian,
    BigEndian
  } machByteOrder = (*((uint8_T *) &one) == 1U) ? LittleEndian : BigEndian;
  switch (machByteOrder) {
   case LittleEndian:
    {
      nanF.wordL.wordLuint = 0xFFC00000U;
      break;
    }

   case BigEndian:
    {
      nanF.wordL.wordLuint = 0x7FFFFFFFU;
      break;
    }
  }

  return nanF.wordL.wordLreal;
}
```

Listed in the project but not available here: Logical/Source/UDP/LibAsUDP1_ST.typ, Logical/Source/UDP/LibAsUDP1_ST.var
